Yaskawa INFORM job: u_incl_braAB0TRJ0.JBI

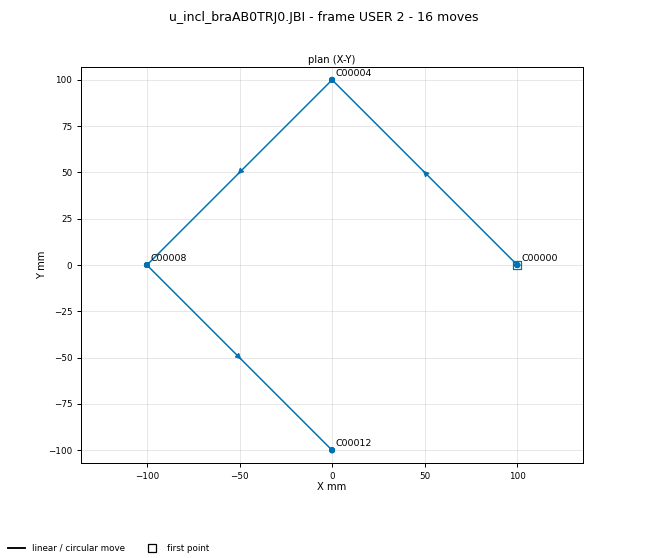
[picture p0: tool path of u_incl_braAB0TRJ0.JBI in frame USER 2, 16 of 16 moves have a stored position in this frame; points joined in program order, loops and branches not executed]
/JOB
//NAME u_incl_braAB0TRJ0
///FOLDERNAME DEMO
//POS
///NPOS 16,0,16,0,0,0
///USER 2
///TOOL 7
///POSTYPE USER
///RECTAN
///RCONF 1,0,0,0,0,0,0,0,0,0,0,0,0,0,0,0,0,0,0,0,0,0,0,0
C00000=100.000,0.000,20.000,-180.0000,20.0125,-180.0000
C00001=100.000,0.000,20.000,159.9875,0.0000,-180.0000
C00002=100.000,0.000,20.000,180.0000,-20.0125,-180.0000
C00003=100.000,0.000,20.000,-159.9875,-0.0000,-180.0000
C00004=0.000,100.000,20.000,-159.9875,-0.0000,-90.0000
C00005=0.000,100.000,20.000,-180.0000,20.0125,-90.0000
C00006=0.000,100.000,20.000,159.9875,0.0000,-90.0000
C00007=0.000,100.000,20.000,180.0000,-20.0125,-90.0000
C00008=-100.000,0.000,20.000,-180.0000,-20.0125,-0.0000
C00009=-100.000,0.000,20.000,-159.9875,0.0000,-0.0000
C00010=-100.000,0.000,20.000,-180.0000,20.0125,-0.0000
C00011=-100.000,0.000,20.000,159.9875,-0.0000,-0.0000
C00012=0.000,-100.000,20.000,159.9875,0.0000,-270.0000
C00013=0.000,-100.000,20.000,180.0000,-20.0125,-270.0000
C00014=0.000,-100.000,20.000,-159.9875,-0.0000,-270.0000
C00015=0.000,-100.000,20.000,-180.0000,20.0125,-270.0000
///TOOL 0
///POSTYPE ANGLE
///ANGLE
EC00000=20.0125,180.0000
EC00001=0.0000,180.0000
EC00002=-20.0125,180.0000
EC00003=-0.0000,180.0000
EC00004=-0.0000,90.0000
EC00005=20.0125,90.0000
EC00006=0.0000,90.0000
EC00007=-20.0125,90.0000
EC00008=-20.0125,0.0000
EC00009=0.0000,0.0000
EC00010=20.0125,0.0000
EC00011=-0.0000,0.0000
EC00012=0.0000,270.0000
EC00013=-20.0125,270.0000
EC00014=-0.0000,270.0000
EC00015=20.0125,270.0000
//INST
///DATE 2022/04/08 11:28
///COMM
///ATTR SC,RW,RJ
////FRAME USER 2
///GROUP1 RB1
///GROUP2 ST1
NOP
SPEED V=10.0
SMOVL C00000 +MOVJ EC00000
SMOVL C00001 +MOVJ EC00001
SMOVL C00002 +MOVJ EC00002
SMOVL C00003 +MOVJ EC00003
SMOVL C00004 +MOVJ EC00004
SMOVL C00005 +MOVJ EC00005
SMOVL C00006 +MOVJ EC00006
SMOVL C00007 +MOVJ EC00007
SMOVL C00008 +MOVJ EC00008
SMOVL C00009 +MOVJ EC00009
SMOVL C00010 +MOVJ EC00010
SMOVL C00011 +MOVJ EC00011
SMOVL C00012 +MOVJ EC00012
SMOVL C00013 +MOVJ EC00013
SMOVL C00014 +MOVJ EC00014
SMOVL C00015 +MOVJ EC00015
END
